{attribute 'linkalways'} 
{attribute 'no_explicit_call' := 'This FB is a CLASS and must be accessed using methods or properties'}
{attribute 'enable_dynamic_creation'}
FUNCTION_BLOCK _TcVnPoint EXTENDS AliasDatatypeBase
VAR
	localData : TcVnPoint;
	activeData : REFERENCE TO TcVnPoint REF= localData;
	aliasBaseDatatype : _TcVnPoint2_DINT;
END_VAR

PROPERTY PUBLIC Address : PVOID
GET
Address := ADR(activeData);
END_GET
END_PROPERTY

METHOD PUBLIC ClearReference
VAR_INPUT
END_VAR
activeData REF= localData;
SetBaseDatatypeReference();
END_METHOD

METHOD PUBLIC Clone : I_Datatype
VAR
    pClone : POINTER TO _TcVnPoint;
END_VAR
pClone := __NEW(_TcVnPoint);
Clone := pClone^;
END_METHOD

METHOD FB_init : BOOL
VAR_INPUT
	bInitRetains : BOOL; // if TRUE, the retain variables are initialized (warm start / cold start)
	bInCopyCode : BOOL;  // if TRUE, the instance afterwards gets moved into the copy code (online change)
	//InitialValue : TcVnPoint; // if possible, not all values can be initialized
END_VAR
//localData := InitialValue; // if possible, not all values can be initialized
SetBaseDatatypeReference();
AddBaseDatatype(aliasBaseDatatype);
END_METHOD

PROPERTY PUBLIC Identifier : T_MAXSTRING
GET
Identifier := 'TcVnPoint';
END_GET
END_PROPERTY

METHOD PUBLIC MakeReferenceTo
VAR_INPUT
	ReferenceTarget : REFERENCE TO TcVnPoint;
END_VAR
activeData REF= ReferenceTarget;
SetBaseDatatypeReference();
END_METHOD

METHOD PROTECTED SetBaseDatatypeReference
VAR_INPUT
END_VAR
aliasBaseDatatype.MakeReferenceTo(activeData);
END_METHOD

PROPERTY PUBLIC Size : UDINT
GET
Size := SIZEOF(activeData);
END_GET
END_PROPERTY

METHOD TryMakeReferenceTo : BOOL
VAR_INPUT
	Target : I_Datatype;
END_VAR
VAR
	targetAsAlias : I_AliasDatatype;
	pTargetData : POINTER TO TcVnPoint;
END_VAR
IF NOT Target.TryResolveAsAliasDatatype(targetAsAlias) THEN
	RETURN;
END_IF

IF targetAsAlias.Identifier <> Identifier THEN
	RETURN;
END_IF

pTargetData := Target.Address;
activeData REF= pTargetData^;
SetBaseDatatypeReference();
TryMakeReferenceTo := TRUE;
END_METHOD

PROPERTY PUBLIC Value : REFERENCE TO TcVnPoint
GET
Value REF= activeData;
END_GET
END_PROPERTY

END_FUNCTION_BLOCK

(* stored: Version 1.1.0.1, ProductVersion 3.1.4024.13
   POU _TcVnPoint: Id {a4ccf06c-6bc7-0aec-1535-586fa788586b}, SpecialFunc None
   Folder Core: Id {00585a07-0779-0785-26f3-e71d8c83a6a1}
   Folder Protected: Id {b2ffc132-4834-0133-2437-7527d549de34}
   Folder Customize: Id {21f3ffa3-4474-0724-0a76-8c41c84f1053}
   Folder Constructor: Id {1e92e7af-c59a-0ba3-3abc-906fdeec800b}
   Property Address: Id {0c90b533-653d-0d57-3534-71572b04fd92}
   Get Get: Id {48b13a09-bcd6-0cc5-16bc-4fa837c2770b}
   Method ClearReference: Id {3b450e53-6433-0381-13d0-424847aed257}
   Method Clone: Id {3c801c61-f04a-074a-2175-ed34f33da1b6}
   Method FB_init: Id {a4de7f8a-811c-0bfa-1047-d9bceeb57af3}
   Property Identifier: Id {56fe04f2-6850-0b29-0a96-3e8801cd021f}
   Get Get: Id {1891e168-78cd-0924-1279-d6ef3b2c5e34}
   Method MakeReferenceTo: Id {93e86fef-bfd6-0b39-194b-36597bca52d2}
   Method SetBaseDatatypeReference: Id {91ae98d4-56dc-019c-367c-9d8805adcff3}
   Property Size: Id {9472f4a1-7082-063f-2ef0-6c3ffe19e42d}
   Get Get: Id {74d7a665-ca2a-0c72-38ed-64f626ac9057}
   Method TryMakeReferenceTo: Id {945153c5-49f5-03d1-3002-9ee724a91dad}
   Property Value: Id {bc8f7d92-3566-01a4-2844-96425bc5693f}
   Get Get: Id {8a3e16aa-bca6-0490-3932-de117346d6a4} *)
